(* Logix 5000 project; controller Drives_Line1 1756-L72 rev 20.13; software revision 20.04; part 20 of 21 *)
(* tags used below, declared in another part *)
   Bridle_04 : UDT_Bridle_3M;
   ExitCtrl : UDT_Control_Zone;
   In_Commands : UDT_Commands;
   In_Config : UDT_Config;
   LineCmd : UDT_Commands_Line;
   Pinchroll_3 : UDT_Pinchroll;
   Pinchroll_3_FB_Diff : DINT;
   Pinchroll_3_FB_Update_Valid : BOOL;
   Pinchroll_3_FBCounts_mm : DINT;
   Pinchroll_3_Max_FB_Counts : DINT;
   Pinchroll_3_Rev_mm : REAL;
   TaskInterval_ms : DINT;
   TestConfig_Pinchroll_3 : UDT_Config_Pinch;
   Winder : UDT_Winder;
   zConfigFromMaster : BOOL;
   zPi : REAL;
   zPinchroll_3_EncRes : DINT;
   zSimulation : BOOL;

PROGRAM P21_Pinchroll_3   (* main routine R00_Main *)
VAR
   ABS_01 : FBD_MATH_ADVANCED;
   BAND_01 : FBD_BOOLEAN_AND := (In1 := 1, In3 := 1, In4 := 1, In5 := 1, In6 := 1, In7 := 1, In8 := 1);
   BAND_02 : FBD_BOOLEAN_AND := (In3 := 1, In4 := 1, In5 := 1, In6 := 1, In7 := 1, In8 := 1);
   BAND_03 : FBD_BOOLEAN_AND := (In3 := 1, In4 := 1, In5 := 1, In6 := 1, In7 := 1, In8 := 1);
   BAND_04 : FBD_BOOLEAN_AND := (In3 := 1, In4 := 1, In5 := 1, In6 := 1, In7 := 1, In8 := 1);
   BAND_05 : FBD_BOOLEAN_AND := (In3 := 1, In4 := 1, In5 := 1, In6 := 1, In7 := 1, In8 := 1);
   BNOT_01 : FBD_BOOLEAN_NOT := (Out := 1);
   BNOT_02 : FBD_BOOLEAN_NOT := (Out := 1);
   BNOT_06 : FBD_BOOLEAN_NOT := (Out := 1);
   BOR_01 : FBD_BOOLEAN_OR;
   FGEN_01 : FUNCTION_GENERATOR := (XY1Size := 1);
   IO_State_Pinch_3 : INT := 6;
   IO_State_Tmp_Pinch_3 : INT := 24576;
   LES_01 : FBD_COMPARE := (SourceB := 0.001, Dest := 1);
   MUL_01 : FBD_MATH := (SourceB := 1145.9155);
   MUL_25 : FBD_MATH := (SourceB := 1145.9155);
   NEG_01 : FBD_MATH_ADVANCED := (Source := 0.1, Dest := -0.1);
   Pinchroll_3_EncRes : DINT := 1024;
   Pinchroll_3_FB_Count_Old : DINT;
   Pinchroll_3_JLossCrvSpd : REAL[21];
   Pinchroll_3_LossCrvTrq_Pct : REAL[21];
   Pinchroll_3_Max_FBcounts : DINT;
   Pinchroll_3_RPMPerMPS : REAL := 1145.9155;
   RLIM_01 : RATE_LIMITER := (IncRate := 0.1, DecRate := 0.1, RTSTime := 1, DeltaT := 0.05);
   SCRV_02 : S_CURVE := (Initialize := 1, AbsAlgRamp := 1, AccelRate := 0.2, DecelRate := 0.2, JerkRate := 0.2, RTSTime := 1, DeltaT := 0.04);
   SSUM_01 : SELECTED_SUMMER := (Gain1 := 1.0, Gain2 := 1.0, Gain3 := 1.0, Select3 := 1, Gain4 := 1.0, Gain5 := 1.0, Gain6 := 1.0, Gain7 := 1.0, Gain8 := 1.0);
   SSUM_05 : SELECTED_SUMMER := (In1 := 0.1, Gain1 := 1.0, In2 := -0.1, Gain2 := 1.0, Gain3 := 1.0, Select3 := 1, Gain4 := 1.0, Gain5 := 1.0, Gain6 := 1.0, Gain7 := 1.0, Gain8 := 1.0);
   SSUM_06 : SELECTED_SUMMER := (Gain1 := 1.0, Select1 := 1, Gain2 := 1.0, Gain3 := 1.0, Gain4 := 1.0, Gain5 := 1.0, Gain6 := 1.0, Gain7 := 1.0, Gain8 := 1.0);
   SUB_01 : FBD_MATH;
   TofReset : TIMER := (PRE := 1000, ACC := 1000);
   TonNoResponse : TIMER := (PRE := 2500);
   zPinchroll_3_Max_rev : REAL := 1500.0;
END_VAR

ROUTINE R00_Main   (* ladder *)
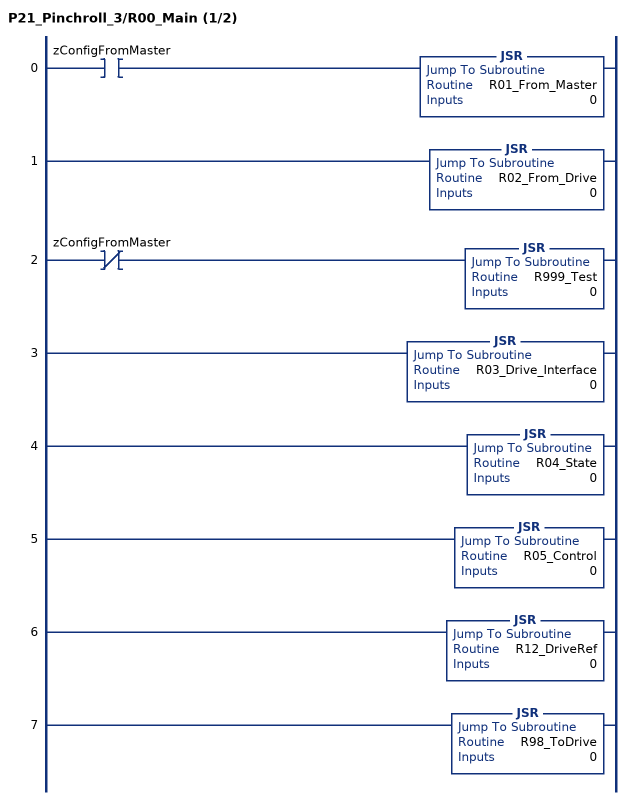
   0: XIC(zConfigFromMaster)JSR(R01_From_Master,0);
   1: JSR(R02_From_Drive,0);
   2: XIO(zConfigFromMaster)JSR(R999_Test,0);
   3: JSR(R03_Drive_Interface,0);
   4: JSR(R04_State,0);
   5: JSR(R05_Control,0);
   6: JSR(R12_DriveRef,0);
   7: JSR(R98_ToDrive,0);
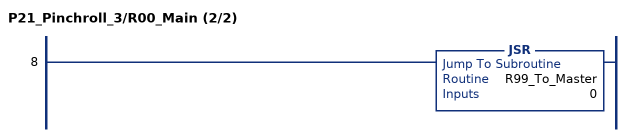
   8: JSR(R99_To_Master,0);
END_ROUTINE

ROUTINE R01_From_Master   (* ladder *)
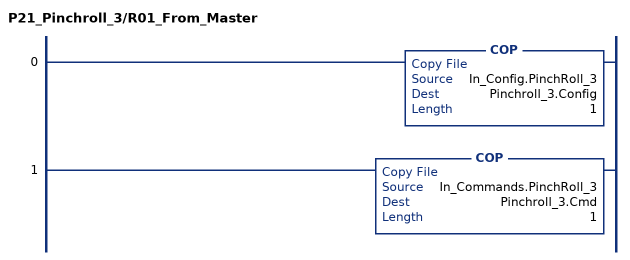
   0: COP(In_Config.PinchRoll_3,Pinchroll_3.Config,1);
   1: COP(In_Commands.PinchRoll_3,Pinchroll_3.Cmd,1);
END_ROUTINE

ROUTINE R02_From_Drive   (* ladder *)
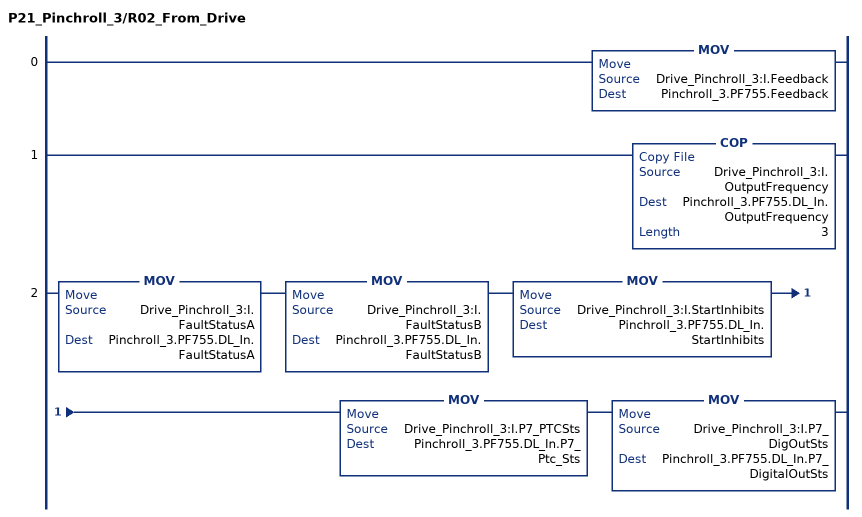
   0: MOV(Drive_Pinchroll_3:I.Feedback,Pinchroll_3.PF755.Feedback);
   1: COP(Drive_Pinchroll_3:I.OutputFrequency,Pinchroll_3.PF755.DL_In.OutputFrequency,3);
   2: MOV(Drive_Pinchroll_3:I.FaultStatusA,Pinchroll_3.PF755.DL_In.FaultStatusA)MOV(Drive_Pinchroll_3:I.FaultStatusB,Pinchroll_3.PF755.DL_In.FaultStatusB)MOV(Drive_Pinchroll_3:I.StartInhibits,Pinchroll_3.PF755.DL_In.StartInhibits)MOV(Drive_Pinchroll_3:I.P7_PTCSts,Pinchroll_3.PF755.DL_In.P7_Ptc_Sts)MOV(Drive_Pinchroll_3:I.P7_DigOutSts,Pinchroll_3.PF755.DL_In.P7_DigitalOutSts);
END_ROUTINE

ROUTINE R03_Drive_Interface   (* ladder *)
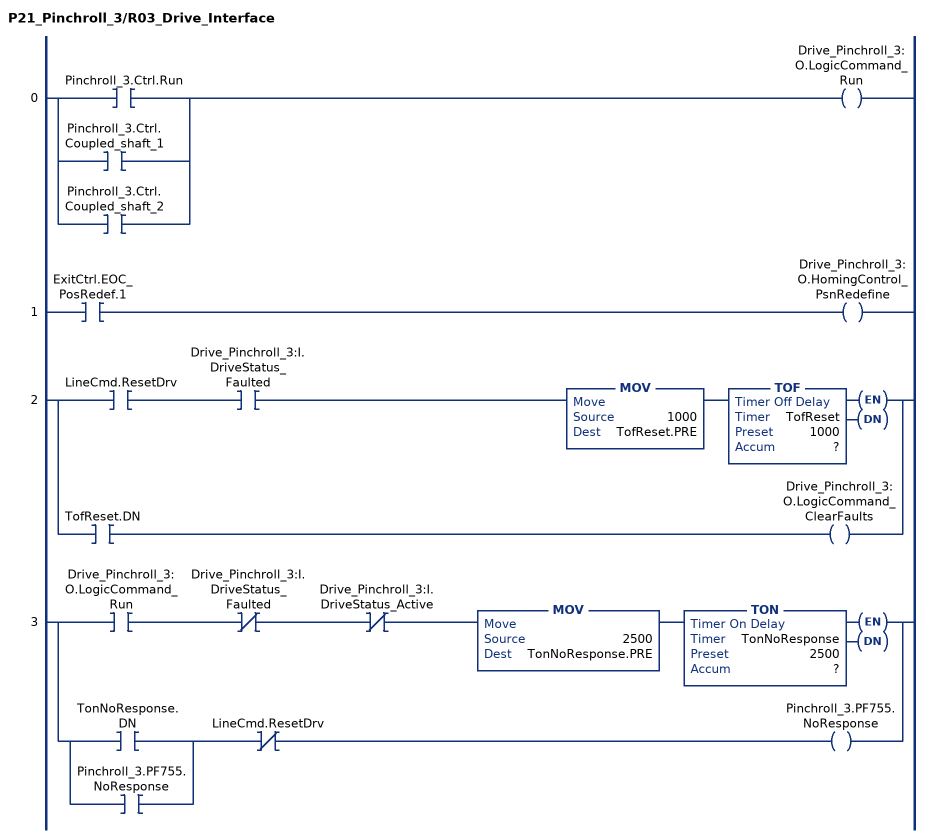
   0: [XIC(Pinchroll_3.Ctrl.Run) ,XIC(Pinchroll_3.Ctrl.Coupled_shaft_1) ,XIC(Pinchroll_3.Ctrl.Coupled_shaft_2) ]OTE(Drive_Pinchroll_3:O.LogicCommand_Run);
   1: XIC(ExitCtrl.EOC_PosRedef.1)OTE(Drive_Pinchroll_3:O.HomingControl_PsnRedefine);
   2: [XIC(LineCmd.ResetDrv) XIC(Drive_Pinchroll_3:I.DriveStatus_Faulted) MOV(1000,TofReset.PRE) TOF(TofReset,?,?) ,XIC(TofReset.DN) OTE(Drive_Pinchroll_3:O.LogicCommand_ClearFaults) ];
   3: [XIC(Drive_Pinchroll_3:O.LogicCommand_Run) XIO(Drive_Pinchroll_3:I.DriveStatus_Faulted) XIO(Drive_Pinchroll_3:I.DriveStatus_Active) MOV(2500,TonNoResponse.PRE) TON(TonNoResponse,?,?) ,[XIC(TonNoResponse.DN) ,XIC(Pinchroll_3.PF755.NoResponse) ] XIO(LineCmd.ResetDrv) OTE(Pinchroll_3.PF755.NoResponse) ];
END_ROUTINE

ROUTINE R04_State   (* ladder *)
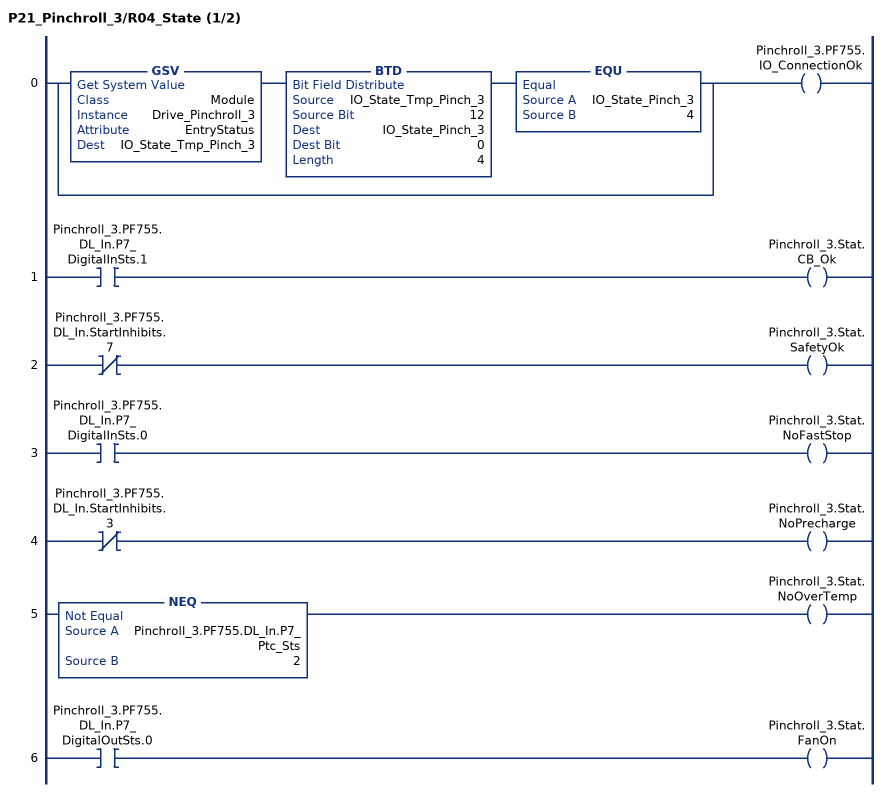
   0: [GSV(Module,Drive_Pinchroll_3,EntryStatus,IO_State_Tmp_Pinch_3) BTD(IO_State_Tmp_Pinch_3,12,IO_State_Pinch_3,0,4) EQU(IO_State_Pinch_3,4) ,]OTE(Pinchroll_3.PF755.IO_ConnectionOk);
   1: XIC(Pinchroll_3.PF755.DL_In.P7_DigitalInSts.1)OTE(Pinchroll_3.Stat.CB_Ok);
   2: XIO(Pinchroll_3.PF755.DL_In.StartInhibits.7)OTE(Pinchroll_3.Stat.SafetyOk);
   3: XIC(Pinchroll_3.PF755.DL_In.P7_DigitalInSts.0)OTE(Pinchroll_3.Stat.NoFastStop);
   4: XIO(Pinchroll_3.PF755.DL_In.StartInhibits.3)OTE(Pinchroll_3.Stat.NoPrecharge);
   5: NEQ(Pinchroll_3.PF755.DL_In.P7_Ptc_Sts,2)OTE(Pinchroll_3.Stat.NoOverTemp);
   6: XIC(Pinchroll_3.PF755.DL_In.P7_DigitalOutSts.0)OTE(Pinchroll_3.Stat.FanOn);
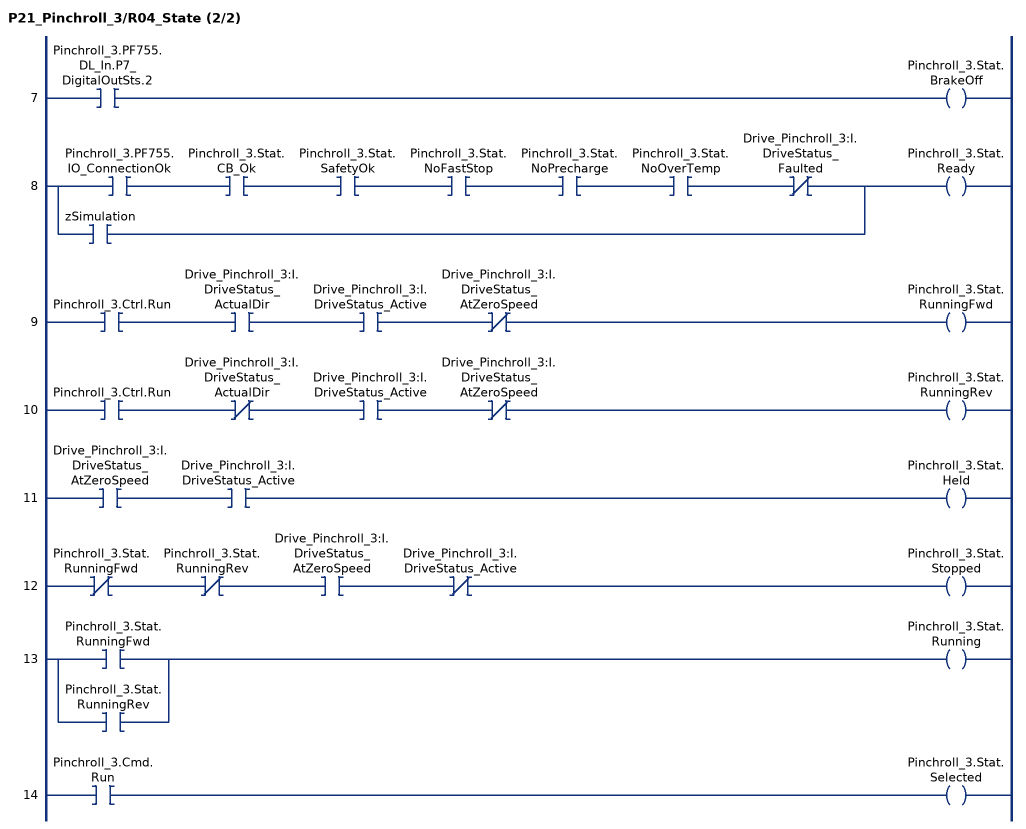
   7: XIC(Pinchroll_3.PF755.DL_In.P7_DigitalOutSts.2)OTE(Pinchroll_3.Stat.BrakeOff);
   8: [XIC(Pinchroll_3.PF755.IO_ConnectionOk) XIC(Pinchroll_3.Stat.CB_Ok) XIC(Pinchroll_3.Stat.SafetyOk) XIC(Pinchroll_3.Stat.NoFastStop) XIC(Pinchroll_3.Stat.NoPrecharge) XIC(Pinchroll_3.Stat.NoOverTemp) XIO(Drive_Pinchroll_3:I.DriveStatus_Faulted) ,XIC(zSimulation) ]OTE(Pinchroll_3.Stat.Ready);
   9: XIC(Pinchroll_3.Ctrl.Run)XIC(Drive_Pinchroll_3:I.DriveStatus_ActualDir)XIC(Drive_Pinchroll_3:I.DriveStatus_Active)XIO(Drive_Pinchroll_3:I.DriveStatus_AtZeroSpeed)OTE(Pinchroll_3.Stat.RunningFwd);
   10: XIC(Pinchroll_3.Ctrl.Run)XIO(Drive_Pinchroll_3:I.DriveStatus_ActualDir)XIC(Drive_Pinchroll_3:I.DriveStatus_Active)XIO(Drive_Pinchroll_3:I.DriveStatus_AtZeroSpeed)OTE(Pinchroll_3.Stat.RunningRev);
   11: XIC(Drive_Pinchroll_3:I.DriveStatus_AtZeroSpeed)XIC(Drive_Pinchroll_3:I.DriveStatus_Active)OTE(Pinchroll_3.Stat.Held);
   12: XIO(Pinchroll_3.Stat.RunningFwd)XIO(Pinchroll_3.Stat.RunningRev)XIC(Drive_Pinchroll_3:I.DriveStatus_AtZeroSpeed)XIO(Drive_Pinchroll_3:I.DriveStatus_Active)OTE(Pinchroll_3.Stat.Stopped);
   13: [XIC(Pinchroll_3.Stat.RunningFwd) ,XIC(Pinchroll_3.Stat.RunningRev) ]OTE(Pinchroll_3.Stat.Running);
   14: XIC(Pinchroll_3.Cmd.Run)OTE(Pinchroll_3.Stat.Selected);
END_ROUTINE

ROUTINE R05_Control   (* ladder *)
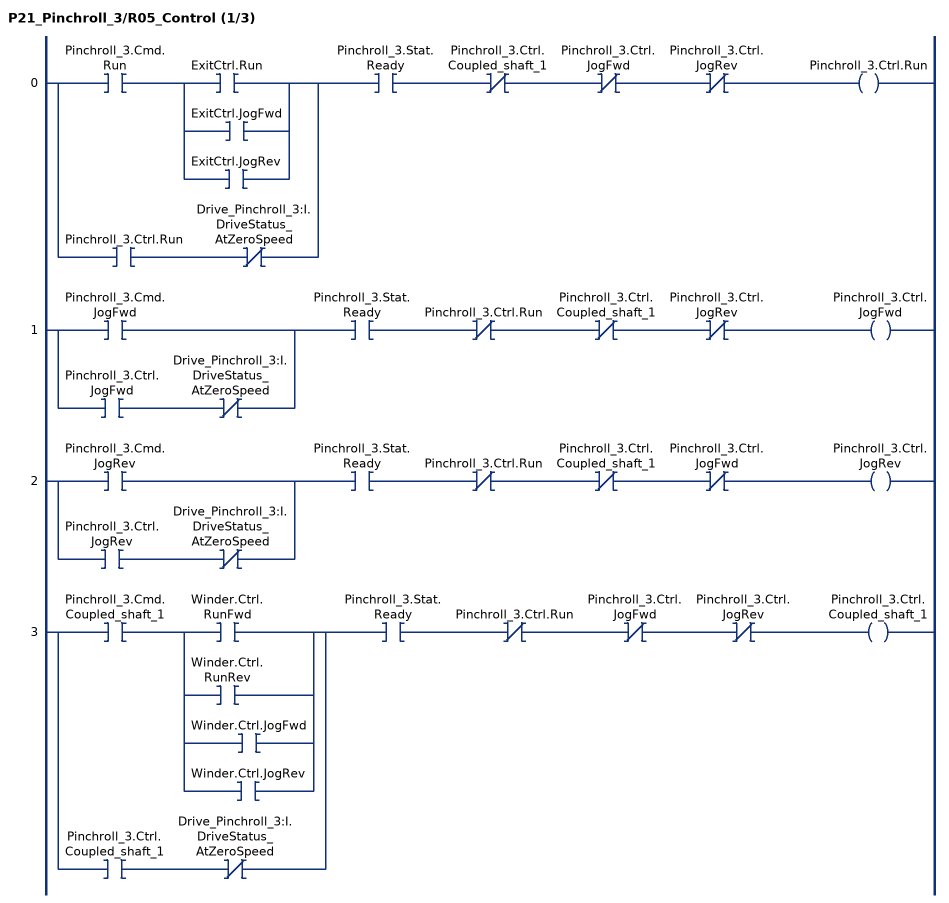
   0: [XIC(Pinchroll_3.Cmd.Run) [XIC(ExitCtrl.Run) ,XIC(ExitCtrl.JogFwd) ,XIC(ExitCtrl.JogRev) ] ,XIC(Pinchroll_3.Ctrl.Run) XIO(Drive_Pinchroll_3:I.DriveStatus_AtZeroSpeed) ]XIC(Pinchroll_3.Stat.Ready)XIO(Pinchroll_3.Ctrl.Coupled_shaft_1)XIO(Pinchroll_3.Ctrl.JogFwd)XIO(Pinchroll_3.Ctrl.JogRev)OTE(Pinchroll_3.Ctrl.Run);
   1: [XIC(Pinchroll_3.Cmd.JogFwd) ,XIC(Pinchroll_3.Ctrl.JogFwd) XIO(Drive_Pinchroll_3:I.DriveStatus_AtZeroSpeed) ]XIC(Pinchroll_3.Stat.Ready)XIO(Pinchroll_3.Ctrl.Run)XIO(Pinchroll_3.Ctrl.Coupled_shaft_1)XIO(Pinchroll_3.Ctrl.JogRev)OTE(Pinchroll_3.Ctrl.JogFwd);
   2: [XIC(Pinchroll_3.Cmd.JogRev) ,XIC(Pinchroll_3.Ctrl.JogRev) XIO(Drive_Pinchroll_3:I.DriveStatus_AtZeroSpeed) ]XIC(Pinchroll_3.Stat.Ready)XIO(Pinchroll_3.Ctrl.Run)XIO(Pinchroll_3.Ctrl.Coupled_shaft_1)XIO(Pinchroll_3.Ctrl.JogFwd)OTE(Pinchroll_3.Ctrl.JogRev);
   3: [XIC(Pinchroll_3.Cmd.Coupled_shaft_1) [XIC(Winder.Ctrl.RunFwd) ,XIC(Winder.Ctrl.RunRev) ,XIC(Winder.Ctrl.JogFwd) ,XIC(Winder.Ctrl.JogRev) ] ,XIC(Pinchroll_3.Ctrl.Coupled_shaft_1) XIO(Drive_Pinchroll_3:I.DriveStatus_AtZeroSpeed) ]XIC(Pinchroll_3.Stat.Ready)XIO(Pinchroll_3.Ctrl.Run)XIO(Pinchroll_3.Ctrl.JogFwd)XIO(Pinchroll_3.Ctrl.JogRev)OTE(Pinchroll_3.Ctrl.Coupled_shaft_1);
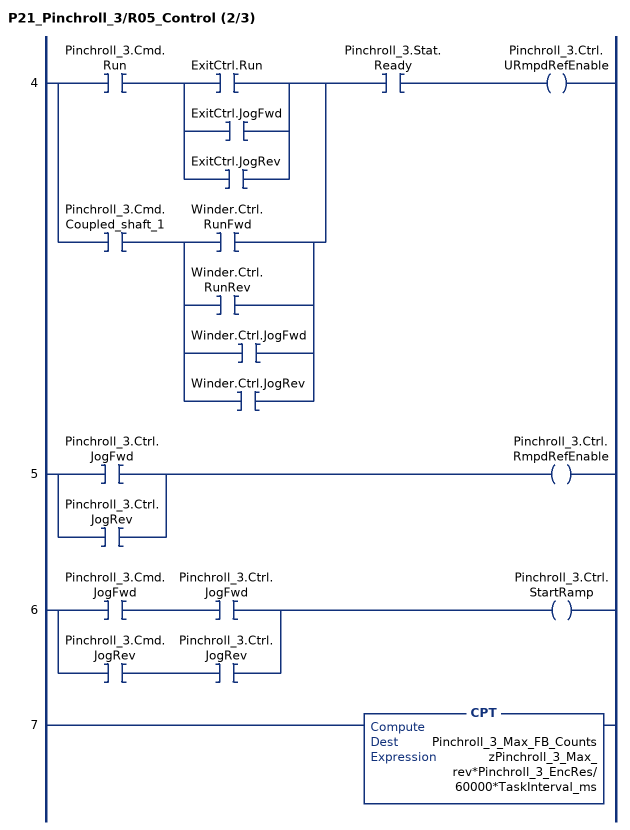
   4: [XIC(Pinchroll_3.Cmd.Run) [XIC(ExitCtrl.Run) ,XIC(ExitCtrl.JogFwd) ,XIC(ExitCtrl.JogRev) ] ,XIC(Pinchroll_3.Cmd.Coupled_shaft_1) [XIC(Winder.Ctrl.RunFwd) ,XIC(Winder.Ctrl.RunRev) ,XIC(Winder.Ctrl.JogFwd) ,XIC(Winder.Ctrl.JogRev) ] ]XIC(Pinchroll_3.Stat.Ready)OTE(Pinchroll_3.Ctrl.URmpdRefEnable);
   5: [XIC(Pinchroll_3.Ctrl.JogFwd) ,XIC(Pinchroll_3.Ctrl.JogRev) ]OTE(Pinchroll_3.Ctrl.RmpdRefEnable);
   6: [XIC(Pinchroll_3.Cmd.JogFwd) XIC(Pinchroll_3.Ctrl.JogFwd) ,XIC(Pinchroll_3.Cmd.JogRev) XIC(Pinchroll_3.Ctrl.JogRev) ]OTE(Pinchroll_3.Ctrl.StartRamp);
   7: CPT(Pinchroll_3_Max_FB_Counts,zPinchroll_3_Max_rev*Pinchroll_3_EncRes/60000*TaskInterval_ms);
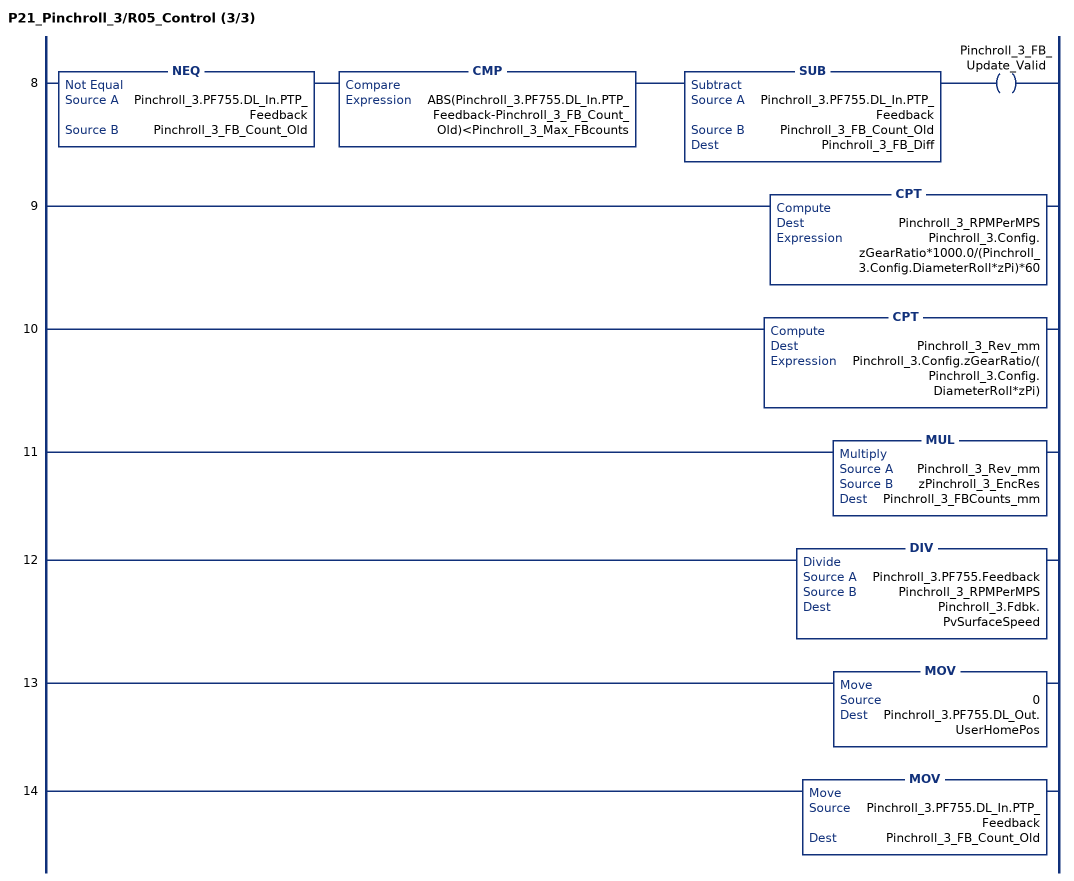
   8: NEQ(Pinchroll_3.PF755.DL_In.PTP_Feedback,Pinchroll_3_FB_Count_Old)CMP(ABS(Pinchroll_3.PF755.DL_In.PTP_Feedback-Pinchroll_3_FB_Count_Old)<Pinchroll_3_Max_FBcounts)SUB(Pinchroll_3.PF755.DL_In.PTP_Feedback,Pinchroll_3_FB_Count_Old,Pinchroll_3_FB_Diff)OTE(Pinchroll_3_FB_Update_Valid);
   9: CPT(Pinchroll_3_RPMPerMPS,Pinchroll_3.Config.zGearRatio*1000.0/(Pinchroll_3.Config.DiameterRoll*zPi)*60);
   10: CPT(Pinchroll_3_Rev_mm,Pinchroll_3.Config.zGearRatio/(Pinchroll_3.Config.DiameterRoll*zPi));
   11: MUL(Pinchroll_3_Rev_mm,zPinchroll_3_EncRes,Pinchroll_3_FBCounts_mm);
   12: DIV(Pinchroll_3.PF755.Feedback,Pinchroll_3_RPMPerMPS,Pinchroll_3.Fdbk.PvSurfaceSpeed);
   13: MOV(0,Pinchroll_3.PF755.DL_Out.UserHomePos);
   14: MOV(Pinchroll_3.PF755.DL_In.PTP_Feedback,Pinchroll_3_FB_Count_Old);
END_ROUTINE

ROUTINE R12_DriveRef   (* function block diagram *)
   SHEET 1   // Select run speed reference
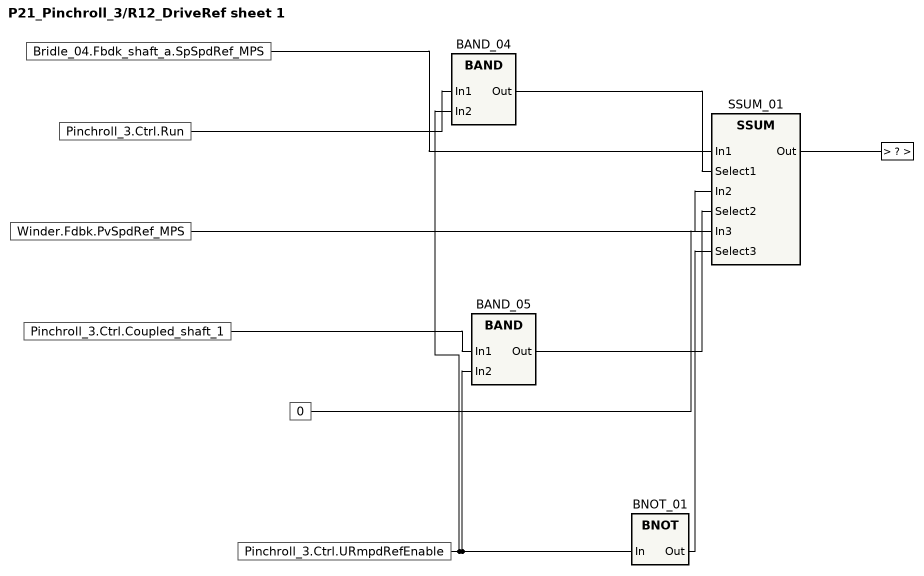
   BAND_04 : BAND(In1 := Pinchroll_3.Ctrl.Run, In2 := Pinchroll_3.Ctrl.URmpdRefEnable);
   BAND_05 : BAND(In1 := Pinchroll_3.Ctrl.Coupled_shaft_1, In2 := Pinchroll_3.Ctrl.URmpdRefEnable);
   BNOT_01 : BNOT(In := Pinchroll_3.Ctrl.URmpdRefEnable);
   SSUM_01 : SSUM(In1 := Bridle_04.Fbdk_shaft_a.SpSpdRef_MPS, Select1 := BAND_04.Out, In2 := Winder.Fdbk.PvSpdRef_MPS, Select2 := BAND_05.Out, In3 := 0, Select3 := BNOT_01.Out);
   WIRE(?) := SSUM_01.Out;
   SHEET 2   // Select jog reference
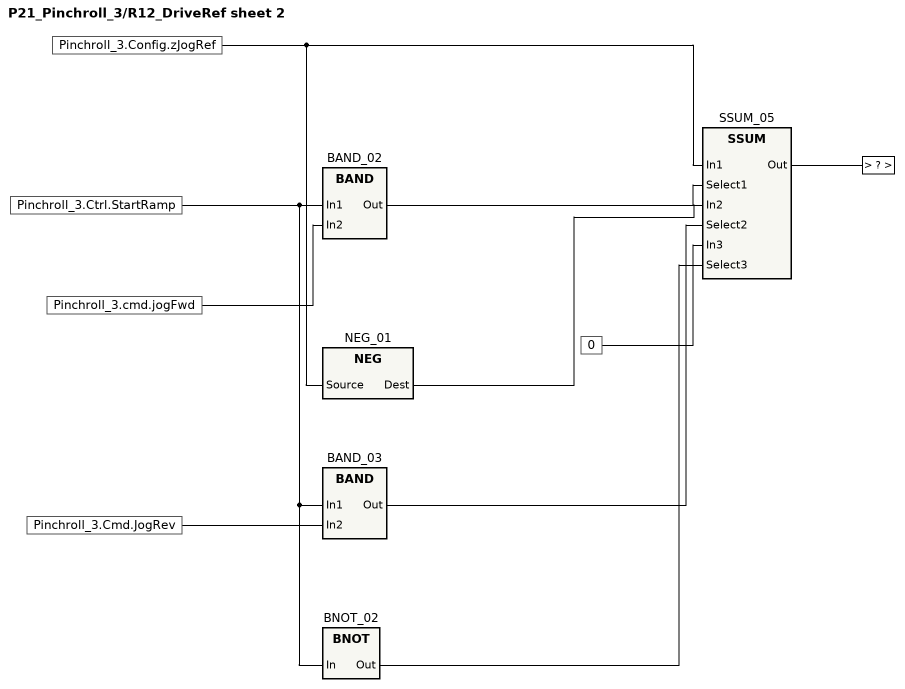
   BAND_02 : BAND(In1 := Pinchroll_3.Ctrl.StartRamp, In2 := Pinchroll_3.cmd.jogFwd);
   NEG_01 : NEG(Source := Pinchroll_3.Config.zJogRef);
   BAND_03 : BAND(In1 := Pinchroll_3.Ctrl.StartRamp, In2 := Pinchroll_3.Cmd.JogRev);
   BNOT_02 : BNOT(In := Pinchroll_3.Ctrl.StartRamp);
   SSUM_05 : SSUM(In1 := Pinchroll_3.Config.zJogRef, Select1 := BAND_02.Out, In2 := NEG_01.Dest, Select2 := BAND_03.Out, In3 := 0, Select3 := BNOT_02.Out);
   WIRE(?) := SSUM_05.Out;
   SHEET 3   // S-Curve
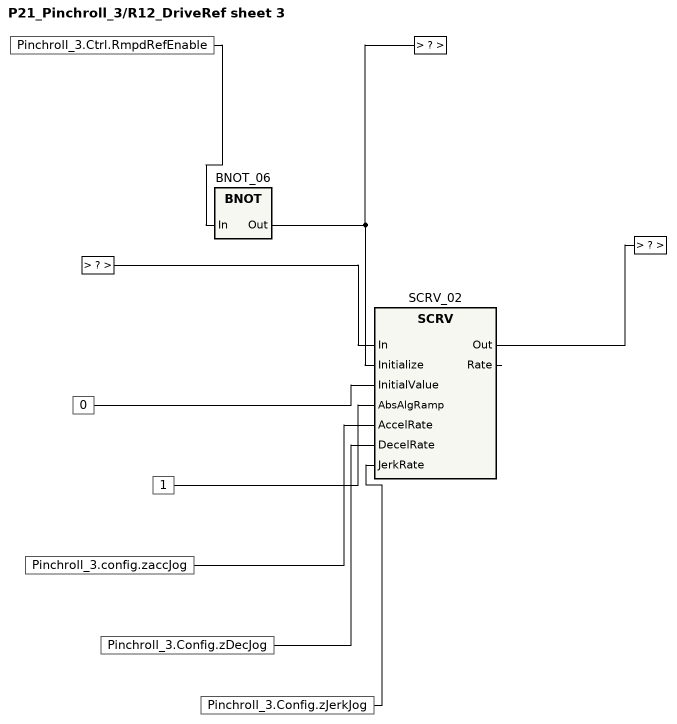
   BNOT_06 : BNOT(In := Pinchroll_3.Ctrl.RmpdRefEnable);
   WIRE(?) := BNOT_06.Out;
   SCRV_02 : SCRV(In := WIRE(?), Initialize := BNOT_06.Out, InitialValue := 0, AbsAlgRamp := 1, AccelRate := Pinchroll_3.config.zaccJog, DecelRate := Pinchroll_3.Config.zDecJog, JerkRate := Pinchroll_3.Config.zJerkJog);   // unwired pins: Rate
   WIRE(?) := SCRV_02.Out;
   SHEET 4   // Select final speed reference
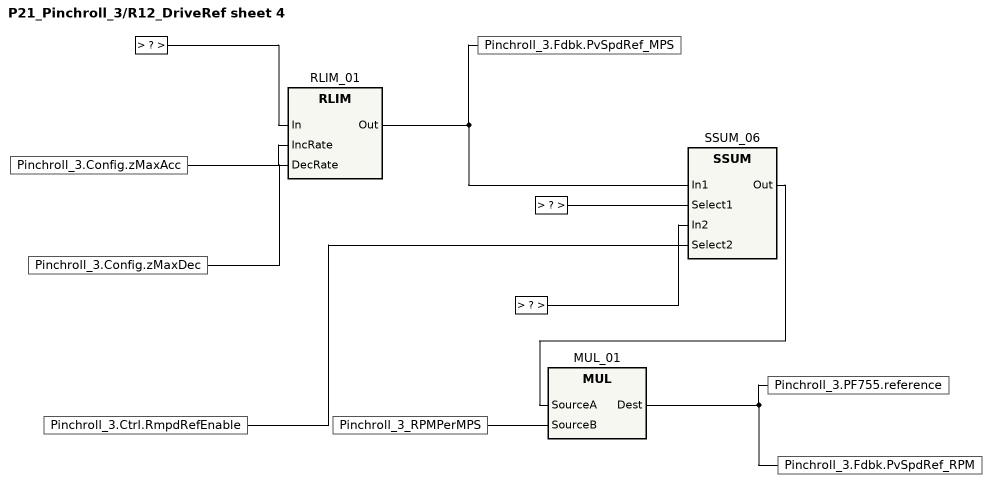
   RLIM_01 : RLIM(In := WIRE(?), IncRate := Pinchroll_3.Config.zMaxAcc, DecRate := Pinchroll_3.Config.zMaxDec);
   Pinchroll_3.Fdbk.PvSpdRef_MPS := RLIM_01.Out;
   SSUM_06 : SSUM(In1 := RLIM_01.Out, Select1 := WIRE(?), In2 := WIRE(?), Select2 := Pinchroll_3.Ctrl.RmpdRefEnable);
   MUL_01 : MUL(SourceA := SSUM_06.Out, SourceB := Pinchroll_3_RPMPerMPS);
   Pinchroll_3.PF755.reference := MUL_01.Dest;
   Pinchroll_3.Fdbk.PvSpdRef_RPM := MUL_01.Dest;
   SHEET 5   // Speed reference synchronized
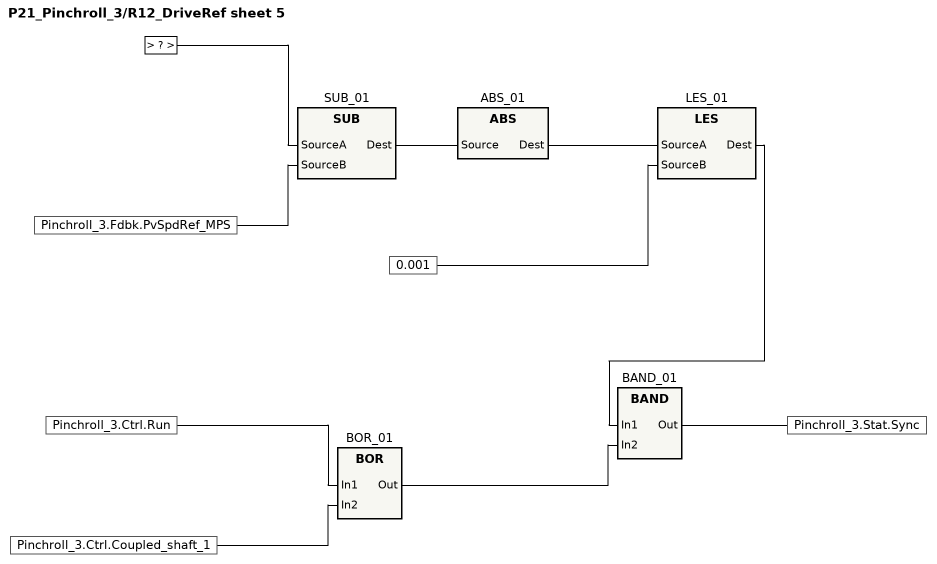
   SUB_01 : SUB(SourceA := WIRE(?), SourceB := Pinchroll_3.Fdbk.PvSpdRef_MPS);
   BOR_01 : BOR(In1 := Pinchroll_3.Ctrl.Run, In2 := Pinchroll_3.Ctrl.Coupled_shaft_1);
   ABS_01 : ABS(Source := SUB_01.Dest);
   LES_01 : LES(SourceA := ABS_01.Dest, SourceB := 0.001);
   BAND_01 : BAND(In1 := LES_01.Dest, In2 := BOR_01.Out);
   Pinchroll_3.Stat.Sync := BAND_01.Out;
   SHEET 6   // Friction compensation
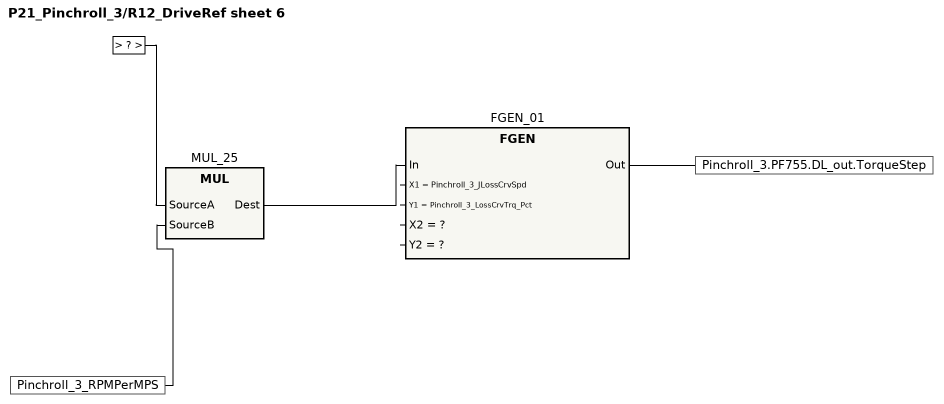
   MUL_25 : MUL(SourceA := WIRE(?), SourceB := Pinchroll_3_RPMPerMPS);
   FGEN_01 : FGEN(In := MUL_25.Dest, X1 := Pinchroll_3_JLossCrvSpd, Y1 := Pinchroll_3_LossCrvTrq_Pct, X2 := ?, Y2 := ?);
   Pinchroll_3.PF755.DL_out.TorqueStep := FGEN_01.Out;
END_ROUTINE

ROUTINE R98_ToDrive   (* ladder *)
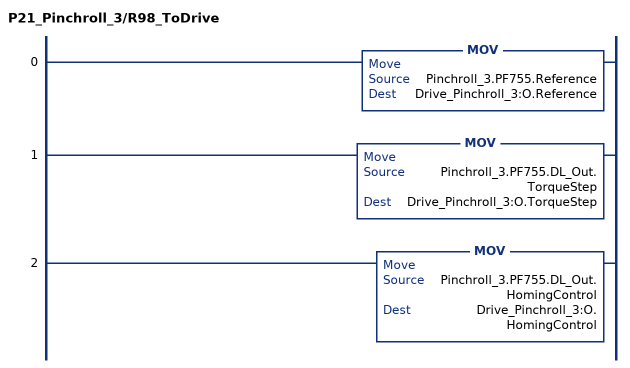
   0: MOV(Pinchroll_3.PF755.Reference,Drive_Pinchroll_3:O.Reference);
   1: MOV(Pinchroll_3.PF755.DL_Out.TorqueStep,Drive_Pinchroll_3:O.TorqueStep);
   2: MOV(Pinchroll_3.PF755.DL_Out.HomingControl,Drive_Pinchroll_3:O.HomingControl);
END_ROUTINE

ROUTINE R999_Test   (* ladder *)
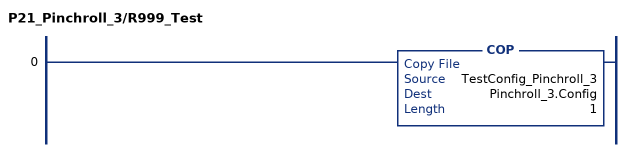
   0: COP(TestConfig_Pinchroll_3,Pinchroll_3.Config,1);
END_ROUTINE
